(*
SPDX-FileCopyrightText: © 2026 Oleksandr Tiutyk <trofimich@gmail.com>
SPDX-License-Identifier: MIT
License: https://opensource.org/license/mit
*)

FUNCTION_BLOCK ABSTRACT EventLoggerMessage EXTENDS TOF_Core.Object
VAR
	{attribute 'OPC.UA.DA':='0'}
	_ClassName : STRING := __POUNAME();
	
	{attribute 'OPC.UA.DA':='0'}
	_Created : BOOL;
	{attribute 'OPC.UA.DA':='0'}
	_MessageSourceInfo : Tc3_EventLogger.FB_TcSourceInfo;
	{attribute 'OPC.UA.DA':='0'}
    _Message : Tc3_EventLogger.FB_TcMessage; 	
END_VAR

PROPERTY ABSTRACT EventEntry : TcEventEntry
GET
END_GET
END_PROPERTY

//!<param name="bInCopyCode">if TRUE, the exit method is called for exiting an instance that is copied afterwards (online change).</param>

METHOD FB_exit : BOOL
VAR_INPUT
	bInCopyCode : BOOL; 
END_VAR
IF _Created THEN
	_Message.Release();
END_IF
END_METHOD

PROPERTY Guid : Global.GUID
GET
Guid := _MessageSourceInfo.guid;
END_GET
SET
_MessageSourceInfo.guid := Guid;
END_SET
END_PROPERTY

{attribute 'monitoring' := 'call'}
PROPERTY Id : UDINT
GET
Id := _MessageSourceInfo.nId;
END_GET
SET
_MessageSourceInfo.nId := Id;
END_SET
END_PROPERTY

METHOD PROTECTED InternalSend
VAR_IN_OUT CONSTANT
	jsonData : STRING(1000);
END_VAR
VAR
	result : HRESULT;
	standardException : TOF_Core.StandardException;
END_VAR
IF NOT _Created THEN
	result := _Message.CreateEx(EventEntry, _MessageSourceInfo);
 
	IF result <> Tc3_Module.S_OK THEN
		standardException.Throw(NamespaceName, ClassName, __POUNAME(), __POSITION(), TOF_Core.WideStrings.Concat255("Message ", TO_WSTRING(ClassName), ": FB_TcMessage.CreateEx failed with HRESULT = ", TO_WSTRING(result)));
	ELSE
		_Created := TRUE;
	END_IF
END_IF

result := _Message.SetJsonAttribute(jsonData);

IF result <> Tc3_Module.S_OK THEN
	standardException.Throw(NamespaceName, ClassName, __POUNAME(), __POSITION(), TOF_Core.WideStrings.Concat255("Message ", TO_WSTRING(ClassName), ": FB_TcMessage.SetJsonAttribute failed with HRESULT = ", TO_WSTRING(result)));
END_IF

result := _Message.Send(0); 

IF result <> Tc3_Module.S_OK THEN
	standardException.Throw(NamespaceName, ClassName, __POUNAME(), __POSITION(), TOF_Core.WideStrings.Concat255("Message ", TO_WSTRING(ClassName), ": FB_TcMessage.Send failed with HRESULT = ", TO_WSTRING(result)));
END_IF
END_METHOD

METHOD PROTECTED InternalTrySend : BOOL
VAR_IN_OUT CONSTANT
	jsonData : STRING(1000);
END_VAR
VAR
	result : HRESULT;
END_VAR
IF NOT _Created THEN
	result := _Message.CreateEx(EventEntry, _MessageSourceInfo);
 
	IF result <> Tc3_Module.S_OK THEN
		RETURN;
	ELSE
		_Created := TRUE;
	END_IF
END_IF

result := _Message.SetJsonAttribute(jsonData);

IF result <> Tc3_Module.S_OK THEN
	RETURN;
END_IF

result := _Message.Send(0); 

IF result <> Tc3_Module.S_OK THEN
	RETURN;
END_IF

InternalTrySend := TRUE;
END_METHOD

{attribute 'monitoring' := 'call'}
PROPERTY SelfSize : ULINT
GET
SelfSize := XSIZEOF(THIS^);
END_GET
END_PROPERTY

{attribute 'monitoring' := 'call'}
PROPERTY SourceName : STRING(255)
GET
SourceName := _MessageSourceInfo.sName;
END_GET
SET
_MessageSourceInfo.sName := SourceName;
END_SET
END_PROPERTY

END_FUNCTION_BLOCK

(* stored: Version 1.1.0.1
   POU EventLoggerMessage: Id {17965dca-217f-4194-b078-823fd63f7465}, SpecialFunc None
   Folder Internal methods: Id {eba39033-b704-48a2-b308-5a1dc901e2dd}
   Property EventEntry: Id {3bf5bc66-fdae-43a5-9ae6-35e04c7302f4}
   Get Get: Id {aaa564d6-f819-43f4-9a0c-f0cfd7ae244b}
   Method FB_exit: Id {fa58c06e-47d0-416d-864c-c44235c7aff8}
   Property Guid: Id {9c28cd55-faa8-4da5-9e84-ea471d98a80c}
   Get Get: Id {de728f70-08bd-416f-bb35-e2ce63ebdf73}
   Set Set: Id {360da14b-66c2-43eb-9d6d-2b05285f40fb}
   Property Id: Id {bb50ba90-8ebd-420f-81ff-d125c6bea821}
   Get Get: Id {18a33dba-1bd9-427b-882f-d36044a6b0fd}
   Set Set: Id {775131c0-7d3c-4801-a794-f914a663029b}
   Method InternalSend: Id {39dacc1d-08e3-4179-94e3-1bf57bb57d58}
   Method InternalTrySend: Id {f4c68b09-4d21-4204-9c94-e88baef1faea}
   Property SelfSize: Id {91cf2cb2-f8a5-4793-b434-4f172abcdbb8}
   Get Get: Id {25f71848-b7bd-4205-afe6-b1c67420251d}
   Property SourceName: Id {2c04cbbf-d187-4935-b54b-eb7d5e9ce04f}
   Get Get: Id {3aa005db-9ea5-4b6c-ada6-1b8c73e81e61}
   Set Set: Id {3c46a52c-f83e-45a0-bfa9-fa822dca2e0b} *)
